{attribute addProperty BoxType "EP6002-0002-0016"}
{attribute addProperty Id "StatusAT %I*WORD1621Data_InAT %I*ARRAY[0 ..21] OF USINT176220"}
{attribute addProperty CRC "3615481419"}
{attribute addProperty SizeInBites "192"}
{attribute addProperty SizeInBytes "24"}
TYPE COM_Inputs_Channel_4EE430B6 :
STRUCT
	{attribute addProperty Name "Status"}
	Status AT %I* : WORD;
	{attribute addProperty Name "Data_In"}
	Data_In AT %I* : ARRAY[0 ..21] OF USINT;
END_STRUCT
END_TYPE

(* stored: Version 1.2.0.0, ProductVersion 3.1.4024.9
   DUT COM_Inputs_Channel_4EE430B6: Id {4492469d-850d-42d8-9be5-c9a6cf1caf8e} *)
